FUNCTION_BLOCK StationSample EXTENDS Process
VAR
	_OperationTime : TIME := T#1S;
	Operation : TON;
	State: INT;
END_VAR

{analysis -2}

METHOD Abort : BOOL
VAR_INPUT
END_VAR
SUPER^();

Abort := TRUE;
_Complete := FALSE;
_Empty := TRUE;
_Operating := FALSE;
_Ready := TRUE;
StationMovers := State := 0;
END_METHOD

METHOD Cycle : HRESULT
VAR
	CycleResult : HRESULT;
END_VAR
Cycle := S_OK;
IF _isProcess THEN
	Operation.IN := _HasMover;
	IF NOT Operation.IN THEN
		_TimeInProcess := Operation.ET;
	END_IF
ELSE
	CASE State OF
		0:
			IF _HasMover THEN
				_Operating := TRUE;
				_Empty := FALSE;
				_Ready := FALSE;
				Operation.IN := TRUE;
				State := 1;
			END_IF
		1:
			IF Operation.Q THEN
				_Complete := TRUE;
				IF StationMovers = 0 THEN
					_HasMover := FALSE;
					Operation.IN := FALSE;
				END_IF
				State := 2;
			END_IF
		2:
			_Complete := FALSE;
			_Empty := TRUE;
			_Operating := FALSE;
			_Ready := TRUE;
			State := 0;
		ELSE
			Cycle := E_FAIL;
	END_CASE	
END_IF

Operation(PT := _OperationTime);

CycleResult := SUPER^.Cycle();
stInfo.StationProcessTime := _OperationTime;

IF CycleResult = E_FAIL THEN
	Cycle := E_FAIL;
END_IF
END_METHOD

PROPERTY TempPropTime : time
GET
TempPropTime := _OperationTime;
END_GET
SET
_OperationTime := TempPropTime;
END_SET
END_PROPERTY

END_FUNCTION_BLOCK

(* stored: Version 1.1.0.1, ProductVersion 3.1.4026.11
   POU StationSample: Id {5d12cef2-4f81-4470-ba05-8f124fe21580}, SpecialFunc None
   Method Abort: Id {21e0d1b2-4f5f-428f-96cf-1000dff3cb8d}
   Method Cycle: Id {b831bddf-8042-4785-99f9-40cdea1773f4}
   Property TempPropTime: Id {4928f043-1047-466d-92d5-fb5212ce41c4}
   Get Get: Id {73c0c3b5-10dd-44f7-bbc4-d091c37d6ab8}
   Set Set: Id {2b0a9403-c0bf-4baf-becb-7504692464bc} *)
